FUNCTION_BLOCK FB_InterfaceIO IMPLEMENTS ITF_Cell
VAR_INPUT

END_VAR
VAR_OUTPUT
END_VAR


	// Ausgang :engine          AT %IX0.0:        BOOL; 
//Eingänge
//A5Q_Bestuckung AT %QX27.4 : BOOL;
//A5Q_Startfreigabe AT %QX27.5 : BOOL;
//A5Q_Entnahme AT %QX27.6 : BOOL;
//A5Q_Standby AT %QX27.7 : BOOL;
//A5Q_NOT_Aus_Befehl AT %QX28.0 : BOOL;

//INPUTS  A5 Station Variabel : 5V Von Arduino

//A5I_Bestuckbereit_o1 AT %IX43.2 : BOOL;  
//A5I_Arbeitet_o2 AT %IX43.3 : BOOL;
//A5I_Fertig_o3 AT %IX43.4 : BOOL;
//A5I_Storung_o5 AT %IX43.5 : BOOL;
//A5I_NOT_Halt_o6 AT %IX43.6 : BOOL;
//A5I_Pro_Standby_o7 AT %IX43.7 : BOOL;
//A5I_Pro_Standby_o8 AT %IX44.0 : BOOL;
VAR
m_bEmergencyOff AT %I* : BOOL;
m_bEmergencyStop AT %I* : BOOL;
m_bFinished AT %I* : BOOL;
m_bRunning AT %I* : BOOL;
m_bLoadPos  AT %I* : BOOL; 
m_bUnloadPos  AT %I* : BOOL; 
m_bStandby AT %I* : BOOL;
m_bStartable AT %I* : BOOL;
m_bSoftError AT %I* : BOOL;
// Ausgang :engine          AT %QX0.0:        BOOL; 
// Ausgänge
m_bToEmergencyOff AT %Q* : BOOL;
m_bToEmergencyStop AT %Q* : BOOL;
m_bMoveToLoadPos AT %Q* : BOOL;
m_bMoveToUnloadPos AT %Q* : BOOL;
m_bToStandby AT %Q* : BOOL;
m_bStart AT %Q* : BOOL;

END_VAR

// Logik des Interfaces in diesem Fall zurücksetzen der Ausgänge nach erreichen des Ziels 
// Aus Zustandsmaschine Löschen ggf. ??
//IF m_bEmergencyOff THEN
//m_bToEmergencyOff := FALSE;
//END_IF

//IF m_bEmergencyStop THEN
//m_bToEmergencyStop := FALSE;
//END_IF

IF m_bLoadPos THEN
	m_bMoveToLoadPos := FALSE;
END_IF

IF m_bUnloadPos THEN
	m_bMoveToUnloadPos := FALSE;
END_IF

IF m_bStandby THEN
	m_bToStandby := FALSE;
END_IF

IF m_bRunning THEN
	m_bStart := FALSE;
END_IF

METHOD GetEmergencyOff : BOOL
VAR_INPUT
END_VAR
GetEmergencyOff := m_bEmergencyOff;
END_METHOD

METHOD GetEmergencyStop : BOOL
VAR_INPUT
END_VAR
GetEmergencyStop := m_bEmergencyStop;
END_METHOD

METHOD GetFinished : BOOL
VAR_INPUT
END_VAR
GetFinished := m_bFinished;
END_METHOD

METHOD GetIsRunning : BOOL
VAR_INPUT
END_VAR
GetIsRunning := m_bRunning;
END_METHOD

METHOD GetLoadPos : BOOL
VAR_INPUT
END_VAR
GetLoadPos := m_bLoadPos;
END_METHOD

METHOD GetStandby : BOOL
VAR_INPUT
END_VAR
GetStandby := m_bStandby;
END_METHOD

METHOD GetStartable : BOOL
VAR_INPUT
END_VAR
GetStartable := m_bStartable;
END_METHOD

METHOD GetUnloadPos : BOOL
VAR_INPUT
END_VAR
GetUnloadPos := m_bUnloadPos;
END_METHOD

METHOD SetEmergencyOff : BOOL
VAR_INPUT
	b :BOOL;
END_VAR

m_bToEmergencyOff := b;
SetEmergencyOff:=b;
END_METHOD

METHOD SetEmergencyStop : BOOL
VAR_INPUT
	b :BOOL;
END_VAR
m_bToEmergencyStop :=b;

SetEmergencyStop := b;
END_METHOD

METHOD SetMoveToLoad : BOOL
VAR_INPUT
	b :BOOL;
END_VAR
m_bMoveToLoadPos := b;

SetMoveToLoad := b;
END_METHOD

METHOD SetMoveToUnload : BOOL
VAR_INPUT
	b :BOOL;
END_VAR
m_bMoveToUnloadPos := b;

SetMoveToUnload := b;
END_METHOD

METHOD SetStandby : BOOL
VAR_INPUT
	b :BOOL;
END_VAR
m_bToStandby := b;

SetStandby := b;
END_METHOD

METHOD SetStart : BOOL
VAR_INPUT
	b :BOOL;
END_VAR
m_bStart := b;

SetStart := b;
END_METHOD

END_FUNCTION_BLOCK

(* stored: Version 1.1.0.1, ProductVersion 3.1.4024.0
   POU FB_InterfaceIO: Id {83fe8b06-4652-45a6-a9e4-2627299933a8}, SpecialFunc None
   Method GetEmergencyOff: Id {7821cdbf-3d5a-425d-8d9d-bad88f016439}
   Method GetEmergencyStop: Id {bc16d24b-9bba-451b-af80-d92660a4b4cb}
   Method GetFinished: Id {0e3ffbfb-88e2-4179-ad72-16ac2c0a96a5}
   Method GetIsRunning: Id {b319ccd4-b513-4e21-9898-63f6e4b613c7}
   Method GetLoadPos: Id {3df13fee-7983-4f01-93d3-717ad048bbed}
   Method GetStandby: Id {4fa0ae63-0a00-4266-b5b4-5ce5afe13f62}
   Method GetStartable: Id {b66c34dc-28bd-480b-8f8a-525c5603dae9}
   Method GetUnloadPos: Id {238b264e-f925-431e-870d-21a2ddbe2715}
   Method SetEmergencyOff: Id {e99c93d4-20d9-4179-9dcc-b10ba1a9b07d}
   Method SetEmergencyStop: Id {f71633d7-a533-4cc9-bfed-b0d65910b911}
   Method SetMoveToLoad: Id {3fe18960-198f-44ad-b5fe-5b1794681f1d}
   Method SetMoveToUnload: Id {a0c31b7c-bf1f-4bd0-9650-540c8f9f13d3}
   Method SetStandby: Id {56214aa5-6565-4319-b48b-c36fe0c7f655}
   Method SetStart: Id {180c4627-461a-404c-9905-d7096503dbde} *)
